TYPE ST_HMIDigInputs :
STRUCT
	bHMIEStartCalibration	: BOOL := FALSE; //Start Calibration Bt from HMI
	bHMIEAbortCalibration	: BOOL := FALSE; //Abort Calibration Bt from HMI
	
	bRebootPLC				: BOOL := FALSE; //Reboot PLC bt from HMI
	bShutdownPLC			: BOOL := FALSE; //Shutdown PLC bt from HMI
	
END_STRUCT
END_TYPE

(* stored: Version 1.1.0.1, ProductVersion 3.1.4024.12
   DUT ST_HMIDigInputs: Id {856a834f-0a9d-4c88-8f4f-88b3463c6d1b} *)
